FUNCTION_BLOCK FB_ltCurtains EXTENDS FB_pushBtnNC
VAR
	bLftCurtainFbError 		AT %I* : BOOL;
	bLftCurtainSigOk 		AT %I* : BOOL;
	bRhtCurtainFbError 		AT %I* : BOOL;
	bRhtCurtainSigOk 		AT %I* : BOOL;
	nLftCurtainFbState 		AT %I* : USINT; //States : 1 - Running, 2 - PreOp, 3 - Triggered, 6 - Reset 
	nRhtCurtainFbState 		AT %I* : USINT; //States : 1 - Running, 2 - PreOp, 3 - Triggered, 6 - Reset 
	

	bRhtCurtainEnable	AT %Q* : BOOL;
	bLftCurtainEnable	AT %Q* : BOOL;
	bResetLftCurtainFb 	AT %Q* : BOOL;
	bResetRhtCurtainFb 	AT %Q* : BOOL;
	bMuteCurtains 		AT %Q* : BOOL;
	
	bCurtainsMuted		AT %I* : BOOL;
	
END_VAR

PROPERTY curtainsMuted : BOOL
GET
curtainsMuted := bCurtainsMuted;
END_GET
END_PROPERTY

PROPERTY enableLftCurtain : BOOL
SET
bLftCurtainEnable := enableLftCurtain;
END_SET
END_PROPERTY

PROPERTY enableRhtCurtain : BOOL
SET
bRhtCurtainEnable := enableRhtCurtain;
END_SET
END_PROPERTY

METHOD mute : BOOL
VAR_INPUT
END_VAR
bMuteCurtains := TRUE;
mute := TRUE;
END_METHOD

METHOD reset : BOOL
VAR_INPUT
END_VAR
reset := FALSE;
bResetLftCurtainFb 	:= TRUE;
bResetRhtCurtainFb 	:= TRUE;

(*IF NOT GVL_machine.bLightCurtainsOk THEN
	bResetLftCurtainFb 	:= FALSE;
	bResetRhtCurtainFb 	:= FALSE;
	reset := TRUE;
END_IF*)
END_METHOD

PROPERTY resetLftCurtainFB : BOOL
SET
bResetLftCurtainFb := resetLftCurtainFB;
END_SET
END_PROPERTY

PROPERTY resetRhtCurtainFB : BOOL
SET
bResetRhtCurtainFb := resetRhtCurtainFB;
END_SET
END_PROPERTY

METHOD unmute : BOOL
VAR_INPUT
END_VAR
bMuteCurtains := FALSE;
unmute := TRUE;
END_METHOD

END_FUNCTION_BLOCK

(* stored: Version 1.1.0.1, ProductVersion 3.1.4024.13
   POU FB_ltCurtains: Id {c70223c6-dd8c-4dcf-8286-84cf4bd1fc56}, SpecialFunc None
   Property curtainsMuted: Id {d6533652-449f-468c-a986-c9b568b13f3e}
   Get Get: Id {ed36f076-4f5d-43dd-859e-a121dbdc4e01}
   Property enableLftCurtain: Id {f4723c28-2852-40ee-8052-0951da5c885c}
   Set Set: Id {9ecb6982-d6ca-4bff-979b-3850342c8d7d}
   Property enableRhtCurtain: Id {314778af-c8a9-4f73-bf3a-7a9e4f5f8c0f}
   Set Set: Id {aa90021d-f0c9-4f8d-8e34-70ee05bcd5da}
   Method mute: Id {3beb5be0-d98c-4c48-9772-6e99b4c14dc6}
   Method reset: Id {948fbe5e-3860-4b8d-a512-4f9b0583287f}
   Property resetLftCurtainFB: Id {539bca16-d6bf-47ee-bc3f-6325ddf62a8e}
   Set Set: Id {8266bb6e-bd58-4e61-b133-b0d8af772d9a}
   Property resetRhtCurtainFB: Id {5b5a279c-5b02-4e86-8dd5-21bb4754315b}
   Set Set: Id {1439c6b8-6188-4a43-bd03-11ba90c10ebb}
   Method unmute: Id {23778aa8-2cea-4649-aefe-67f3d76c6b1c} *)
